Yaskawa INFORM job: LTCHGPS1.JBI

/JOB
//NAME LTCHGPS1
//POS
///NPOS 0,0,0,0,0,0
//INST
///DATE 2019/11/21 17:40
///ATTR SC,RW,MC
///GROUP1 RB1,BS1
///GROUP2 ST1
///LVARS 1,0,0,0,0,0,0,0
NOP
'**************************
'** Chang of GAP File    **
'**      MACRO JOB       **
'**for Std. Laser-Tracker**
'**************************
'=== initialize ===
'--- GAP File No -----------
GETARG LB000 IARG#(1)
'
SKILLSND ATTR=3 "LTRACKCH GF:0"
'
END
